// TwinCAT 3 PLC project virtual_plc
// ProgramVersion: 3.1.4024.0
// libraries:
//   Tc2_Standard, * (Beckhoff Automation GmbH)
//   Tc2_System, * (Beckhoff Automation GmbH)
//   Tc3_Module, * (Beckhoff Automation GmbH)
// project tree:
//   GVLs/ GVL.TcGVL
//   / PlcTask.TcTTO
//   POUs/ MAIN.TcPOU, carride.TcPOU, treinrit_program.TcPOU
// real-time tasks:
//   TASK PlcTask: cycle T#10ms, priority 20, ADS port 350

CONFIGURATION virtual_plc
    RESOURCE PLC ON TwinCAT3
        TASK PlcTask(INTERVAL := T#10ms, PRIORITY := 20);
        PROGRAM MAIN WITH PlcTask : MAIN;
        PROGRAM treinrit_program WITH PlcTask : treinrit_program;
    END_RESOURCE
END_CONFIGURATION

// ---- GVLs/GVL.TcGVL
{attribute 'qualified_only'}
VAR_GLOBAL

    //starting signals
    bStartDrive : BOOL := FALSE;
    bStartWalk1 : BOOL := FALSE;
    bStartTrain : BOOL := FALSE;
    bStartWalk2 : BOOL := FALSE;
    InternalStart : BOOL;
	bArrived: BOOL := FALSE;
	
	
    //State machine
    Step : INT := 0;
	train : INT := 0;

    //Info
    sStatus : STRING;
	TravelTime : TIME := T#12S; //treinrit tijd
END_VAR

// ---- POUs/MAIN.TcPOU
PROGRAM MAIN
VAR
     (*Timers*)
    tDriveHomeToStation : TON := (PT := T#15S);   //car ride
    tWalkHomeToStation : TON := (PT := T#10S);    //walking
    tWalkStationToSchool : TON := (PT := T#8S);   // walking
	
	    (* car FB *)
    car : Carride;
	
END_VAR

CASE gvl.Step OF

    0: (* Start at home *)
        gvl.sStatus := 'leaving home, get in the car, driving to station';
        gvl.bStartDrive := TRUE;
        //tDriveHomeToStation(IN := gvl.bStartDrive);
		car(bStart := gvl.bStartDrive, TravelTime := T#12S);

        IF car.bcararrived THEN
            gvl.bStartDrive := FALSE;
            tDriveHomeToStation(IN := FALSE);
            gvl.Step := 5;
        END_IF;


    5: (* Walking from car to train*)
        gvl.sStatus := 'parked the car. Walking to the station.';
        gvl.bStartWalk1 := TRUE;
        tWalkHomeToStation(IN := gvl.bStartWalk1);

        IF tWalkHomeToStation.Q THEN
            gvl.bStartWalk1 := FALSE;
            tWalkHomeToStation(IN := FALSE);
            gvl.Step := 10;
        END_IF;


    10: (* Start train*)
        gvl.sStatus := 'Aarrived at the station. Train leaves.';
        gvl.bStartTrain := TRUE;

        IF gvl.barrived THEN
            gvl.bStartTrain := FALSE;
            gvl.Step := 20;
        END_IF;


    20: (* Walking from train to school *)
        gvl.sStatus := 'Train arrived. Walking to school.';
        gvl.bStartWalk2 := TRUE;
        tWalkStationToSchool(IN := gvl.bStartWalk2);

        IF tWalkStationToSchool.Q THEN
            tWalkStationToSchool(IN := FALSE);
            gvl.bStartWalk2 := FALSE;
            gvl.Step := 30;
        END_IF;


    30: (* Arrived at school *)
        gvl.sStatus := 'arrived at school';


ELSE
    gvl.sStatus := 'ERROR, I am lost.';
END_CASE;

END_PROGRAM

// ---- POUs/carride.TcPOU
FUNCTION_BLOCK carride
VAR_INPUT
    bStart : BOOL;
    TravelTime : TIME;
END_VAR

VAR_OUTPUT
    bcarArrived : BOOL := FALSE;
END_VAR

VAR
	tTimerauto :ton := (PT := T#8S); // timer auto
END_VAR

IF bStart AND NOT gvl.InternalStart THEN
    gvl.InternalStart := TRUE;
    bcarArrived := FALSE;
    tTimerauto(IN := TRUE, PT := TravelTime);
END_IF;

tTimerauto(IN := tTimerauto.IN, PT := TravelTime);


IF tTimerauto.Q THEN
    bcarArrived := TRUE;
    tTimerauto(IN := FALSE);
    gvl.InternalStart := FALSE;
END_IF;

END_FUNCTION_BLOCK

// ---- POUs/treinrit_program.TcPOU
PROGRAM treinrit_program
VAR
	Start: BOOL;
	
	 //Timers
	Timer : TON := (PT := gvl.TravelTime);	//train timer

END_VAR

CASE gvl.train OF

0:
IF gvl.bStartTrain AND NOT gvl.InternalStart THEN
	gvl.train := 5;
END_IF;

5:

  	gvl.InternalStart := TRUE;
    gvl.bArrived := FALSE;
    Timer(in := gvl.bStarttrain);
	
IF Timer.Q THEN
    gvl.bArrived := TRUE;
    Timer(IN := FALSE);
    gvl.InternalStart := FALSE;
END_IF;

END_CASE;

END_PROGRAM
